(*

short summary
=============
This function returns a reference to a π-nana.
The π-nana is created by a pineapple type and a banana type.
The reference points to a π-nana on the stack memory.

legal notes
===========
SPDX-FileCopyrightText: © 2024 ekvip automation GmbH <info@ekvip.de>
SPDX-License-Identifier: Apache-2.0
For details check: Apache-2.0_

.. _Apache-2.0: https://www.apache.org/licenses/LICENSE-2.0

*)
FUNCTION GetAPinanaFromStack :REFERENCE TO Pinana
VAR_INPUT
	(* type of pineapple to create a π-nana from it *)
	pineapple	:PineappleType;
	(* type of banana to create a π-nana from it *)
	banana		:BananaType;
END_VAR
VAR
	(* stack π-nana to refer on it *)
	stackPinana :Pinana;
END_VAR

GetAPinanaFromStack REF= 0;
(* validate parameters *)
RETURN((pineapple = PineappleType.NONE) OR (banana = BananaType.NONE));

(* initialize stack π-nana *)
stackPinana.me := ADR(stackPinana);
stackPinana.pinanaType := (TO_UDINT(pineapple) + TO_UDINT(banana));
stackPinana.variety := TO_STRING(stackPinana.pinanaType);
stackPinana.curve := CalculatePinanaCurvature(stackPinana.pinanaType);
GetAPinanaFromStack REF= stackPinana;

END_FUNCTION

(* stored: Version 1.1.0.1, ProductVersion 3.1.4024.12
   POU GetAPinanaFromStack: Id {0f38c109-bc72-45fb-a285-cbfa8b3312cf}, SpecialFunc None *)
